FUNCTION_BLOCK MaskedSwitch
  (* Standard: 61499-2 *)
  (* Version 0.1, 2017-00-22, hpea485, UOA *)
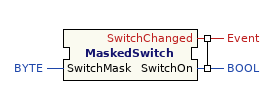
  EVENT_OUTPUT
    SwitchChanged WITH SwitchOn;
  END_EVENT
  VAR_INPUT
    SwitchMask : BYTE;
  END_VAR
  VAR_OUTPUT
    SwitchOn : BOOL;
  END_VAR
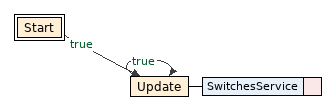
  EC_STATES
    Start;
    Update : SwitchesService;
  END_STATES
  EC_TRANSITIONS
    Start TO Update := true;
    Update TO Update := true;
  END_TRANSITIONS
  ALGORITHM SwitchesService IN C:
int m = (SWITCHES & me->SwitchMask) != 0;
if(m != me->SwitchOn) {
	//switch is pressed
	me->SwitchOn = m;
	me->outputEvents.event.SwitchChanged = 1;
}
  END_ALGORITHM
END_FUNCTION_BLOCK
